// TwinCAT 3 PLC project Test_PLC_1
// ProgramVersion: 3.1.4024.0
// libraries:
//   Tc2_EtherCAT, * (Beckhoff Automation GmbH)
//   Tc2_Standard, * (Beckhoff Automation GmbH)
//   Tc2_System, * (Beckhoff Automation GmbH)
//   Tc3_Mc3PlanarMotion, * (Beckhoff Automation GmbH)
//   Tc3_Module, * (Beckhoff Automation GmbH)
//   Tc3_Physics, * (Beckhoff Automation GmbH)
//   Tc3_XPlanarStandard, * (Beckhoff Automation GmbH)
//   Tc3_XPlanarUtility, * (Beckhoff Automation GmbH)
//   VisuSymbols,3.5.10.0,System
// project tree:
//   DUTs/ ST_MoverParameters.TcDUT
//   / GlobalTextList.TcGTLO, PlcTask.TcTTO, Visualization Manager.TcVMO (not stored)
//   GVLs/ IO.TcGVL
//   POUs/Analytics/ CoeToPlc.TcPOU
//   POUs/ MAIN.TcPOU
//   POUs/xPlanar/ xPlanarControl.TcPOU, xPlanarProgram.TcPOU
//   VISUs/ Visualization.TcVIS
// real-time tasks:
//   TASK Job Task: cycle default, priority 32
//   TASK MC-Task (MET): cycle T#2ms, priority 10, ADS port 521
//   TASK MC-Task (MPT): cycle T#10ms, priority 18, ADS port 531
//   TASK PlcTask: cycle T#10ms, priority 20, ADS port 351
//   TASK XPlanar Task8: cycle T#250us, priority 4, ADS port 352
//   TASK XPlanar Task4: cycle T#250us, priority 6, ADS port 350
//   TASK PlcTask1: cycle T#10ms, priority 14, ADS port 353
// motion (NC):
//   TASK NC-Task 1 SAF: cycle T#2ms, priority 8, ADS port 501
//   TASK NC-Task 1 SVB: cycle T#10ms, priority 16, ADS port 511
//   AXIS Mover a-axis (id 2)
//     OtherSettings: AllowMotionCmdToSlave=true
//     encoder EncType=1
//     drive DrvType=5
//       Analog: TorqueSetpointScale=10, ScaleFactorActTorque=0.1
//       TimeComp: TaskDelayCycles=1
//     controller CtrType=1
//       CtrPara: PriorControlFactor=1
//         Observer: BandWidth=20
//   AXIS Mover b-axis (id 3)
//     OtherSettings: AllowMotionCmdToSlave=true
//     encoder EncType=1
//     drive DrvType=5
//       Analog: TorqueSetpointScale=10, ScaleFactorActTorque=0.1
//       TimeComp: TaskDelayCycles=1
//     controller CtrType=1
//       CtrPara: PriorControlFactor=1
//         Observer: BandWidth=20
//   AXIS Mover c-axis (id 4)
//     OtherSettings: AllowMotionCmdToSlave=true
//     encoder EncType=1
//     drive DrvType=5
//       Analog: TorqueSetpointScale=10, ScaleFactorActTorque=0.1
//       TimeComp: TaskDelayCycles=1
//     controller CtrType=1
//       CtrPara: PriorControlFactor=1
//         Observer: BandWidth=20
//   AXIS Mover x-axis (id 5)
//     OtherSettings: AllowMotionCmdToSlave=true
//     encoder EncType=1
//     drive DrvType=5
//       Analog: TorqueSetpointScale=10, ScaleFactorActTorque=0.1
//       TimeComp: TaskDelayCycles=1
//     controller CtrType=1
//       CtrPara: PriorControlFactor=1
//         Observer: BandWidth=20
//   AXIS Mover y-axis (id 6)
//     OtherSettings: AllowMotionCmdToSlave=true
//     encoder EncType=1
//     drive DrvType=5
//       Analog: TorqueSetpointScale=10, ScaleFactorActTorque=0.1
//       TimeComp: TaskDelayCycles=1
//     controller CtrType=1
//       CtrPara: PriorControlFactor=1
//         Observer: BandWidth=20
//   AXIS Mover z-axis (id 7)
//     OtherSettings: AllowMotionCmdToSlave=true
//     encoder EncType=1
//     drive DrvType=5
//       Analog: TorqueSetpointScale=10, ScaleFactorActTorque=0.1
//       TimeComp: TaskDelayCycles=1
//     controller CtrType=1
//       CtrPara: PriorControlFactor=1
//         Observer: BandWidth=20
// I/O:
//   DEVICE Device 1 (EtherCAT) (disabled), AmsNetId 192.168.5.90.2.1
//     Term 1 (EK1200) [EK1200-5000 EtherCAT Power supply (2A E-Bus)]
//       Term 2 (EL1004) [EL1004 4Ch. Dig. Input 24V, 3ms]
//       Term 3 (EL2004) [EL2004 4Ch. Dig. Output 24V, 0.5A]
//       Term 4 (EL9011) [EL9011 End Terminal]
//   DEVICE Device 4 (EtherCAT) (disabled), AmsNetId 192.168.5.90.7.1
//     Term 5 (APS4322-7000) [APS4322-7000 Drive]
//       Term 6 (APS4322-5000) [APS4322-5000 Feedback]
//     Term 7 (APS4322-7000) [APS4322-7000 Drive]
//       Term 8 (APS4322-5000) [APS4322-5000 Feedback]
// variable links:
//   Device 4 (EtherCAT) <-> TcCOM Objects/XPlanar/Part1/Tile1
//     Term 5 (APS4322-7000)/APS Comm Inputs/CommStatusWord <-> Data Pointer/MoverCommStatusWord
//     Term 5 (APS4322-7000)/APS Comm Inputs/Data {1..4} <-> Data Pointer/MoverCommDataIn[{0..3}]  (4 links)
//     Term 5 (APS4322-7000)/APS Comm Outputs/CommControlWord <-> Data Pointer/MoverCommControlWord
//     Term 5 (APS4322-7000)/APS Comm Outputs/Data 1 <-> Data Pointer/MoverCommDataOut
//     Term 5 (APS4322-7000)/APS Diagdata/DC Link Voltage <-> Data Pointer/DcLinkVoltage
//     Term 5 (APS4322-7000)/APS Diagdata/Power supply current <-> Data Pointer/PowerSupplyCurrent
//     Term 5 (APS4322-7000)/APS Inputs/StatusWord <-> Data Pointer/PowerUnitStatusWord
//     Term 5 (APS4322-7000)/APS Outputs/ControlWord <-> Data Pointer/PowerUnitControlWord
//     Term 5 (APS4322-7000)/APS Outputs/Current D 0X0 <-> Data Pointer/DCurrentSetPoints[0]
//     Term 5 (APS4322-7000)/APS Outputs/Current D 0X1 <-> Data Pointer/DCurrentSetPoints[1]
//     Term 5 (APS4322-7000)/APS Outputs/Current D 0X2 <-> Data Pointer/DCurrentSetPoints[2]
//     Term 5 (APS4322-7000)/APS Outputs/Current D 1X0 <-> Data Pointer/DCurrentSetPoints[6]
//     Term 5 (APS4322-7000)/APS Outputs/Current D 1X1 <-> Data Pointer/DCurrentSetPoints[7]
//     Term 5 (APS4322-7000)/APS Outputs/Current D 1X2 <-> Data Pointer/DCurrentSetPoints[8]
//     Term 5 (APS4322-7000)/APS Outputs/Current D 2X0 <-> Data Pointer/DCurrentSetPoints[12]
//     Term 5 (APS4322-7000)/APS Outputs/Current D 2X1 <-> Data Pointer/DCurrentSetPoints[13]
//     Term 5 (APS4322-7000)/APS Outputs/Current D 2X2 <-> Data Pointer/DCurrentSetPoints[14]
//     Term 5 (APS4322-7000)/APS Outputs/Current D 3X0 <-> Data Pointer/DCurrentSetPoints[18]
//     Term 5 (APS4322-7000)/APS Outputs/Current D 3X1 <-> Data Pointer/DCurrentSetPoints[19]
//     Term 5 (APS4322-7000)/APS Outputs/Current D 3X2 <-> Data Pointer/DCurrentSetPoints[20]
//     Term 5 (APS4322-7000)/APS Outputs/Current D 0Y0 <-> Data Pointer/DCurrentSetPoints[3]
//     Term 5 (APS4322-7000)/APS Outputs/Current D 0Y1 <-> Data Pointer/DCurrentSetPoints[4]
//     Term 5 (APS4322-7000)/APS Outputs/Current D 0Y2 <-> Data Pointer/DCurrentSetPoints[5]
//     Term 5 (APS4322-7000)/APS Outputs/Current D 1Y0 <-> Data Pointer/DCurrentSetPoints[9]
//     Term 5 (APS4322-7000)/APS Outputs/Current D 1Y1 <-> Data Pointer/DCurrentSetPoints[10]
//     Term 5 (APS4322-7000)/APS Outputs/Current D 1Y2 <-> Data Pointer/DCurrentSetPoints[11]
//     Term 5 (APS4322-7000)/APS Outputs/Current D 2Y0 <-> Data Pointer/DCurrentSetPoints[15]
//     Term 5 (APS4322-7000)/APS Outputs/Current D 2Y1 <-> Data Pointer/DCurrentSetPoints[16]
//     Term 5 (APS4322-7000)/APS Outputs/Current D 2Y2 <-> Data Pointer/DCurrentSetPoints[17]
//     Term 5 (APS4322-7000)/APS Outputs/Current D 3Y0 <-> Data Pointer/DCurrentSetPoints[21]
//     Term 5 (APS4322-7000)/APS Outputs/Current D 3Y1 <-> Data Pointer/DCurrentSetPoints[22]
//     Term 5 (APS4322-7000)/APS Outputs/Current D 3Y2 <-> Data Pointer/DCurrentSetPoints[23]
//     Term 5 (APS4322-7000)/APS Outputs/Current Q 0X0 <-> Data Pointer/QCurrentSetPoints[0]
//     Term 5 (APS4322-7000)/APS Outputs/Current Q 0X1 <-> Data Pointer/QCurrentSetPoints[1]
//     Term 5 (APS4322-7000)/APS Outputs/Current Q 0X2 <-> Data Pointer/QCurrentSetPoints[2]
//     Term 5 (APS4322-7000)/APS Outputs/Current Q 1X0 <-> Data Pointer/QCurrentSetPoints[6]
//     Term 5 (APS4322-7000)/APS Outputs/Current Q 1X1 <-> Data Pointer/QCurrentSetPoints[7]
//     Term 5 (APS4322-7000)/APS Outputs/Current Q 1X2 <-> Data Pointer/QCurrentSetPoints[8]
//     Term 5 (APS4322-7000)/APS Outputs/Current Q 2X0 <-> Data Pointer/QCurrentSetPoints[12]
//     Term 5 (APS4322-7000)/APS Outputs/Current Q 2X1 <-> Data Pointer/QCurrentSetPoints[13]
//     Term 5 (APS4322-7000)/APS Outputs/Current Q 2X2 <-> Data Pointer/QCurrentSetPoints[14]
//     Term 5 (APS4322-7000)/APS Outputs/Current Q 3X0 <-> Data Pointer/QCurrentSetPoints[18]
//     Term 5 (APS4322-7000)/APS Outputs/Current Q 3X1 <-> Data Pointer/QCurrentSetPoints[19]
//     Term 5 (APS4322-7000)/APS Outputs/Current Q 3X2 <-> Data Pointer/QCurrentSetPoints[20]
//     Term 5 (APS4322-7000)/APS Outputs/Current Q 0Y0 <-> Data Pointer/QCurrentSetPoints[3]
//     Term 5 (APS4322-7000)/APS Outputs/Current Q 0Y1 <-> Data Pointer/QCurrentSetPoints[4]
//     Term 5 (APS4322-7000)/APS Outputs/Current Q 0Y2 <-> Data Pointer/QCurrentSetPoints[5]
//     Term 5 (APS4322-7000)/APS Outputs/Current Q 1Y0 <-> Data Pointer/QCurrentSetPoints[9]
//     Term 5 (APS4322-7000)/APS Outputs/Current Q 1Y1 <-> Data Pointer/QCurrentSetPoints[10]
//     Term 5 (APS4322-7000)/APS Outputs/Current Q 1Y2 <-> Data Pointer/QCurrentSetPoints[11]
//     Term 5 (APS4322-7000)/APS Outputs/Current Q 2Y0 <-> Data Pointer/QCurrentSetPoints[15]
//     Term 5 (APS4322-7000)/APS Outputs/Current Q 2Y1 <-> Data Pointer/QCurrentSetPoints[16]
//     Term 5 (APS4322-7000)/APS Outputs/Current Q 2Y2 <-> Data Pointer/QCurrentSetPoints[17]
//     Term 5 (APS4322-7000)/APS Outputs/Current Q 3Y0 <-> Data Pointer/QCurrentSetPoints[21]
//     Term 5 (APS4322-7000)/APS Outputs/Current Q 3Y1 <-> Data Pointer/QCurrentSetPoints[22]
//     Term 5 (APS4322-7000)/APS Outputs/Current Q 3Y2 <-> Data Pointer/QCurrentSetPoints[23]
//     Term 5 (APS4322-7000)/APS Outputs/PhiE 0X0 <-> Data Pointer/PhiSetPoints[0]
//     Term 5 (APS4322-7000)/APS Outputs/PhiE 0X1 <-> Data Pointer/PhiSetPoints[1]
//     Term 5 (APS4322-7000)/APS Outputs/PhiE 0X2 <-> Data Pointer/PhiSetPoints[2]
//     Term 5 (APS4322-7000)/APS Outputs/PhiE 1X0 <-> Data Pointer/PhiSetPoints[6]
//     Term 5 (APS4322-7000)/APS Outputs/PhiE 1X1 <-> Data Pointer/PhiSetPoints[7]
//     Term 5 (APS4322-7000)/APS Outputs/PhiE 1X2 <-> Data Pointer/PhiSetPoints[8]
//     Term 5 (APS4322-7000)/APS Outputs/PhiE 2X0 <-> Data Pointer/PhiSetPoints[12]
//     Term 5 (APS4322-7000)/APS Outputs/PhiE 2X1 <-> Data Pointer/PhiSetPoints[13]
//     Term 5 (APS4322-7000)/APS Outputs/PhiE 2X2 <-> Data Pointer/PhiSetPoints[14]
//     Term 5 (APS4322-7000)/APS Outputs/PhiE 3X0 <-> Data Pointer/PhiSetPoints[18]
//     Term 5 (APS4322-7000)/APS Outputs/PhiE 3X1 <-> Data Pointer/PhiSetPoints[19]
//     Term 5 (APS4322-7000)/APS Outputs/PhiE 3X2 <-> Data Pointer/PhiSetPoints[20]
//     Term 5 (APS4322-7000)/APS Outputs/PhiE 0Y0 <-> Data Pointer/PhiSetPoints[3]
//     Term 5 (APS4322-7000)/APS Outputs/PhiE 0Y1 <-> Data Pointer/PhiSetPoints[4]
//     Term 5 (APS4322-7000)/APS Outputs/PhiE 0Y2 <-> Data Pointer/PhiSetPoints[5]
//     Term 5 (APS4322-7000)/APS Outputs/PhiE 1Y0 <-> Data Pointer/PhiSetPoints[9]
//     Term 5 (APS4322-7000)/APS Outputs/PhiE 1Y1 <-> Data Pointer/PhiSetPoints[10]
//     Term 5 (APS4322-7000)/APS Outputs/PhiE 1Y2 <-> Data Pointer/PhiSetPoints[11]
//     Term 5 (APS4322-7000)/APS Outputs/PhiE 2Y0 <-> Data Pointer/PhiSetPoints[15]
//     Term 5 (APS4322-7000)/APS Outputs/PhiE 2Y1 <-> Data Pointer/PhiSetPoints[16]
//     Term 5 (APS4322-7000)/APS Outputs/PhiE 2Y2 <-> Data Pointer/PhiSetPoints[17]
//     Term 5 (APS4322-7000)/APS Outputs/PhiE 3Y0 <-> Data Pointer/PhiSetPoints[21]
//     Term 5 (APS4322-7000)/APS Outputs/PhiE 3Y1 <-> Data Pointer/PhiSetPoints[22]
//     Term 5 (APS4322-7000)/APS Outputs/PhiE 3Y2 <-> Data Pointer/PhiSetPoints[23]
//     Term 5 (APS4322-7000)/Term 6 (APS4322-5000)/FB Inputs/A{0..8 step 2} X-Field <-> Data Pointer/HallSensorFieldsXYZ[{0..12 step 3}]  (5 links)
//     Term 5 (APS4322-7000)/Term 6 (APS4322-5000)/FB Inputs/A{0..8 step 2} Y-Field <-> Data Pointer/HallSensorFieldsXYZ[{1..13 step 3}]  (5 links)
//     Term 5 (APS4322-7000)/Term 6 (APS4322-5000)/FB Inputs/A{0..8 step 2} Z-Field <-> Data Pointer/HallSensorFieldsXYZ[{2..14 step 3}]  (5 links)
//     Term 5 (APS4322-7000)/Term 6 (APS4322-5000)/FB Inputs/B{1..9 step 2} X-Field <-> Data Pointer/HallSensorFieldsXYZ[{15..27 step 3}]  (5 links)
//     Term 5 (APS4322-7000)/Term 6 (APS4322-5000)/FB Inputs/B{1..9 step 2} Y-Field <-> Data Pointer/HallSensorFieldsXYZ[{16..28 step 3}]  (5 links)
//     Term 5 (APS4322-7000)/Term 6 (APS4322-5000)/FB Inputs/B{1..9 step 2} Z-Field <-> Data Pointer/HallSensorFieldsXYZ[{17..29 step 3}]  (5 links)
//     Term 5 (APS4322-7000)/Term 6 (APS4322-5000)/FB Inputs/C{0..8 step 2} X-Field <-> Data Pointer/HallSensorFieldsXYZ[{30..42 step 3}]  (5 links)
//     Term 5 (APS4322-7000)/Term 6 (APS4322-5000)/FB Inputs/C{0..8 step 2} Y-Field <-> Data Pointer/HallSensorFieldsXYZ[{31..43 step 3}]  (5 links)
//     Term 5 (APS4322-7000)/Term 6 (APS4322-5000)/FB Inputs/C{0..8 step 2} Z-Field <-> Data Pointer/HallSensorFieldsXYZ[{32..44 step 3}]  (5 links)
//     Term 5 (APS4322-7000)/Term 6 (APS4322-5000)/FB Inputs/D{1..9 step 2} X-Field <-> Data Pointer/HallSensorFieldsXYZ[{45..57 step 3}]  (5 links)
//     Term 5 (APS4322-7000)/Term 6 (APS4322-5000)/FB Inputs/D{1..9 step 2} Y-Field <-> Data Pointer/HallSensorFieldsXYZ[{46..58 step 3}]  (5 links)
//     Term 5 (APS4322-7000)/Term 6 (APS4322-5000)/FB Inputs/D{1..9 step 2} Z-Field <-> Data Pointer/HallSensorFieldsXYZ[{47..59 step 3}]  (5 links)
//     Term 5 (APS4322-7000)/Term 6 (APS4322-5000)/FB Inputs/E{0..8 step 2} X-Field <-> Data Pointer/HallSensorFieldsXYZ[{60..72 step 3}]  (5 links)
//     Term 5 (APS4322-7000)/Term 6 (APS4322-5000)/FB Inputs/E{0..8 step 2} Y-Field <-> Data Pointer/HallSensorFieldsXYZ[{61..73 step 3}]  (5 links)
//     Term 5 (APS4322-7000)/Term 6 (APS4322-5000)/FB Inputs/E{0..8 step 2} Z-Field <-> Data Pointer/HallSensorFieldsXYZ[{62..74 step 3}]  (5 links)
//     Term 5 (APS4322-7000)/Term 6 (APS4322-5000)/FB Inputs/F{1..9 step 2} X-Field <-> Data Pointer/HallSensorFieldsXYZ[{75..87 step 3}]  (5 links)
//     Term 5 (APS4322-7000)/Term 6 (APS4322-5000)/FB Inputs/F{1..9 step 2} Y-Field <-> Data Pointer/HallSensorFieldsXYZ[{76..88 step 3}]  (5 links)
//     Term 5 (APS4322-7000)/Term 6 (APS4322-5000)/FB Inputs/F{1..9 step 2} Z-Field <-> Data Pointer/HallSensorFieldsXYZ[{77..89 step 3}]  (5 links)
//     Term 5 (APS4322-7000)/Term 6 (APS4322-5000)/FB Inputs/G{0..8 step 2} X-Field <-> Data Pointer/HallSensorFieldsXYZ[{90..102 step 3}]  (5 links)
//     Term 5 (APS4322-7000)/Term 6 (APS4322-5000)/FB Inputs/G{0..8 step 2} Y-Field <-> Data Pointer/HallSensorFieldsXYZ[{91..103 step 3}]  (5 links)
//     Term 5 (APS4322-7000)/Term 6 (APS4322-5000)/FB Inputs/G{0..8 step 2} Z-Field <-> Data Pointer/HallSensorFieldsXYZ[{92..104 step 3}]  (5 links)
//     Term 5 (APS4322-7000)/Term 6 (APS4322-5000)/FB Inputs/H{1..9 step 2} X-Field <-> Data Pointer/HallSensorFieldsXYZ[{105..117 step 3}]  (5 links)
//     Term 5 (APS4322-7000)/Term 6 (APS4322-5000)/FB Inputs/H{1..9 step 2} Y-Field <-> Data Pointer/HallSensorFieldsXYZ[{106..118 step 3}]  (5 links)
//     Term 5 (APS4322-7000)/Term 6 (APS4322-5000)/FB Inputs/H{1..9 step 2} Z-Field <-> Data Pointer/HallSensorFieldsXYZ[{107..119 step 3}]  (5 links)
//     Term 5 (APS4322-7000)/Term 6 (APS4322-5000)/FB Inputs/I{0..8 step 2} X-Field <-> Data Pointer/HallSensorFieldsXYZ[{120..132 step 3}]  (5 links)
//     Term 5 (APS4322-7000)/Term 6 (APS4322-5000)/FB Inputs/I{0..8 step 2} Y-Field <-> Data Pointer/HallSensorFieldsXYZ[{121..133 step 3}]  (5 links)
//     Term 5 (APS4322-7000)/Term 6 (APS4322-5000)/FB Inputs/I{0..8 step 2} Z-Field <-> Data Pointer/HallSensorFieldsXYZ[{122..134 step 3}]  (5 links)
//     Term 5 (APS4322-7000)/Term 6 (APS4322-5000)/FB Inputs/J{1..9 step 2} X-Field <-> Data Pointer/HallSensorFieldsXYZ[{135..147 step 3}]  (5 links)
//     Term 5 (APS4322-7000)/Term 6 (APS4322-5000)/FB Inputs/J{1..9 step 2} Y-Field <-> Data Pointer/HallSensorFieldsXYZ[{136..148 step 3}]  (5 links)
//     Term 5 (APS4322-7000)/Term 6 (APS4322-5000)/FB Inputs/J{1..9 step 2} Z-Field <-> Data Pointer/HallSensorFieldsXYZ[{137..149 step 3}]  (5 links)
//     Term 5 (APS4322-7000)/Term 6 (APS4322-5000)/FB Inputs/Status <-> Data Pointer/FeedbackStatus
//   Device 4 (EtherCAT) <-> TcCOM Objects/XPlanar/Part1/Tile2
//     Term 7 (APS4322-7000)/APS Comm Inputs/CommStatusWord <-> Data Pointer/MoverCommStatusWord
//     Term 7 (APS4322-7000)/APS Comm Inputs/Data {1..4} <-> Data Pointer/MoverCommDataIn[{0..3}]  (4 links)
//     Term 7 (APS4322-7000)/APS Comm Outputs/CommControlWord <-> Data Pointer/MoverCommControlWord
//     Term 7 (APS4322-7000)/APS Comm Outputs/Data 1 <-> Data Pointer/MoverCommDataOut
//     Term 7 (APS4322-7000)/APS Diagdata/DC Link Voltage <-> Data Pointer/DcLinkVoltage
//     Term 7 (APS4322-7000)/APS Diagdata/Power supply current <-> Data Pointer/PowerSupplyCurrent
//     Term 7 (APS4322-7000)/APS Inputs/StatusWord <-> Data Pointer/PowerUnitStatusWord
//     Term 7 (APS4322-7000)/APS Outputs/ControlWord <-> Data Pointer/PowerUnitControlWord
//     Term 7 (APS4322-7000)/APS Outputs/Current D 0X0 <-> Data Pointer/DCurrentSetPoints[0]
//     Term 7 (APS4322-7000)/APS Outputs/Current D 0X1 <-> Data Pointer/DCurrentSetPoints[1]
//     Term 7 (APS4322-7000)/APS Outputs/Current D 0X2 <-> Data Pointer/DCurrentSetPoints[2]
//     Term 7 (APS4322-7000)/APS Outputs/Current D 1X0 <-> Data Pointer/DCurrentSetPoints[6]
//     Term 7 (APS4322-7000)/APS Outputs/Current D 1X1 <-> Data Pointer/DCurrentSetPoints[7]
//     Term 7 (APS4322-7000)/APS Outputs/Current D 1X2 <-> Data Pointer/DCurrentSetPoints[8]
//     Term 7 (APS4322-7000)/APS Outputs/Current D 2X0 <-> Data Pointer/DCurrentSetPoints[12]
//     Term 7 (APS4322-7000)/APS Outputs/Current D 2X1 <-> Data Pointer/DCurrentSetPoints[13]
//     Term 7 (APS4322-7000)/APS Outputs/Current D 2X2 <-> Data Pointer/DCurrentSetPoints[14]
//     Term 7 (APS4322-7000)/APS Outputs/Current D 3X0 <-> Data Pointer/DCurrentSetPoints[18]
//     Term 7 (APS4322-7000)/APS Outputs/Current D 3X1 <-> Data Pointer/DCurrentSetPoints[19]
//     Term 7 (APS4322-7000)/APS Outputs/Current D 3X2 <-> Data Pointer/DCurrentSetPoints[20]
//     Term 7 (APS4322-7000)/APS Outputs/Current D 0Y0 <-> Data Pointer/DCurrentSetPoints[3]
//     Term 7 (APS4322-7000)/APS Outputs/Current D 0Y1 <-> Data Pointer/DCurrentSetPoints[4]
//     Term 7 (APS4322-7000)/APS Outputs/Current D 0Y2 <-> Data Pointer/DCurrentSetPoints[5]
//     Term 7 (APS4322-7000)/APS Outputs/Current D 1Y0 <-> Data Pointer/DCurrentSetPoints[9]
//     Term 7 (APS4322-7000)/APS Outputs/Current D 1Y1 <-> Data Pointer/DCurrentSetPoints[10]
//     Term 7 (APS4322-7000)/APS Outputs/Current D 1Y2 <-> Data Pointer/DCurrentSetPoints[11]
//     Term 7 (APS4322-7000)/APS Outputs/Current D 2Y0 <-> Data Pointer/DCurrentSetPoints[15]
//     Term 7 (APS4322-7000)/APS Outputs/Current D 2Y1 <-> Data Pointer/DCurrentSetPoints[16]
//     Term 7 (APS4322-7000)/APS Outputs/Current D 2Y2 <-> Data Pointer/DCurrentSetPoints[17]
//     Term 7 (APS4322-7000)/APS Outputs/Current D 3Y0 <-> Data Pointer/DCurrentSetPoints[21]
//     Term 7 (APS4322-7000)/APS Outputs/Current D 3Y1 <-> Data Pointer/DCurrentSetPoints[22]
//     Term 7 (APS4322-7000)/APS Outputs/Current D 3Y2 <-> Data Pointer/DCurrentSetPoints[23]
//     Term 7 (APS4322-7000)/APS Outputs/Current Q 0X0 <-> Data Pointer/QCurrentSetPoints[0]
//     Term 7 (APS4322-7000)/APS Outputs/Current Q 0X1 <-> Data Pointer/QCurrentSetPoints[1]
//     Term 7 (APS4322-7000)/APS Outputs/Current Q 0X2 <-> Data Pointer/QCurrentSetPoints[2]
//     Term 7 (APS4322-7000)/APS Outputs/Current Q 1X0 <-> Data Pointer/QCurrentSetPoints[6]
//     Term 7 (APS4322-7000)/APS Outputs/Current Q 1X1 <-> Data Pointer/QCurrentSetPoints[7]
//     Term 7 (APS4322-7000)/APS Outputs/Current Q 1X2 <-> Data Pointer/QCurrentSetPoints[8]
//     Term 7 (APS4322-7000)/APS Outputs/Current Q 2X0 <-> Data Pointer/QCurrentSetPoints[12]
//     Term 7 (APS4322-7000)/APS Outputs/Current Q 2X1 <-> Data Pointer/QCurrentSetPoints[13]
//     Term 7 (APS4322-7000)/APS Outputs/Current Q 2X2 <-> Data Pointer/QCurrentSetPoints[14]
//     Term 7 (APS4322-7000)/APS Outputs/Current Q 3X0 <-> Data Pointer/QCurrentSetPoints[18]
//     Term 7 (APS4322-7000)/APS Outputs/Current Q 3X1 <-> Data Pointer/QCurrentSetPoints[19]
//     Term 7 (APS4322-7000)/APS Outputs/Current Q 3X2 <-> Data Pointer/QCurrentSetPoints[20]
//     Term 7 (APS4322-7000)/APS Outputs/Current Q 0Y0 <-> Data Pointer/QCurrentSetPoints[3]
//     Term 7 (APS4322-7000)/APS Outputs/Current Q 0Y1 <-> Data Pointer/QCurrentSetPoints[4]
//     Term 7 (APS4322-7000)/APS Outputs/Current Q 0Y2 <-> Data Pointer/QCurrentSetPoints[5]
//     Term 7 (APS4322-7000)/APS Outputs/Current Q 1Y0 <-> Data Pointer/QCurrentSetPoints[9]
//     Term 7 (APS4322-7000)/APS Outputs/Current Q 1Y1 <-> Data Pointer/QCurrentSetPoints[10]
//     Term 7 (APS4322-7000)/APS Outputs/Current Q 1Y2 <-> Data Pointer/QCurrentSetPoints[11]
//     Term 7 (APS4322-7000)/APS Outputs/Current Q 2Y0 <-> Data Pointer/QCurrentSetPoints[15]
//     Term 7 (APS4322-7000)/APS Outputs/Current Q 2Y1 <-> Data Pointer/QCurrentSetPoints[16]
//     Term 7 (APS4322-7000)/APS Outputs/Current Q 2Y2 <-> Data Pointer/QCurrentSetPoints[17]
//     Term 7 (APS4322-7000)/APS Outputs/Current Q 3Y0 <-> Data Pointer/QCurrentSetPoints[21]
//     Term 7 (APS4322-7000)/APS Outputs/Current Q 3Y1 <-> Data Pointer/QCurrentSetPoints[22]
//     Term 7 (APS4322-7000)/APS Outputs/Current Q 3Y2 <-> Data Pointer/QCurrentSetPoints[23]
//     Term 7 (APS4322-7000)/APS Outputs/PhiE 0X0 <-> Data Pointer/PhiSetPoints[0]
//     Term 7 (APS4322-7000)/APS Outputs/PhiE 0X1 <-> Data Pointer/PhiSetPoints[1]
//     Term 7 (APS4322-7000)/APS Outputs/PhiE 0X2 <-> Data Pointer/PhiSetPoints[2]
//     Term 7 (APS4322-7000)/APS Outputs/PhiE 1X0 <-> Data Pointer/PhiSetPoints[6]
//     Term 7 (APS4322-7000)/APS Outputs/PhiE 1X1 <-> Data Pointer/PhiSetPoints[7]
//     Term 7 (APS4322-7000)/APS Outputs/PhiE 1X2 <-> Data Pointer/PhiSetPoints[8]
//     Term 7 (APS4322-7000)/APS Outputs/PhiE 2X0 <-> Data Pointer/PhiSetPoints[12]
//     Term 7 (APS4322-7000)/APS Outputs/PhiE 2X1 <-> Data Pointer/PhiSetPoints[13]
//     Term 7 (APS4322-7000)/APS Outputs/PhiE 2X2 <-> Data Pointer/PhiSetPoints[14]
//     Term 7 (APS4322-7000)/APS Outputs/PhiE 3X0 <-> Data Pointer/PhiSetPoints[18]
//     Term 7 (APS4322-7000)/APS Outputs/PhiE 3X1 <-> Data Pointer/PhiSetPoints[19]
//     Term 7 (APS4322-7000)/APS Outputs/PhiE 3X2 <-> Data Pointer/PhiSetPoints[20]
//     Term 7 (APS4322-7000)/APS Outputs/PhiE 0Y0 <-> Data Pointer/PhiSetPoints[3]
//     Term 7 (APS4322-7000)/APS Outputs/PhiE 0Y1 <-> Data Pointer/PhiSetPoints[4]
//     Term 7 (APS4322-7000)/APS Outputs/PhiE 0Y2 <-> Data Pointer/PhiSetPoints[5]
//     Term 7 (APS4322-7000)/APS Outputs/PhiE 1Y0 <-> Data Pointer/PhiSetPoints[9]
//     Term 7 (APS4322-7000)/APS Outputs/PhiE 1Y1 <-> Data Pointer/PhiSetPoints[10]
//     Term 7 (APS4322-7000)/APS Outputs/PhiE 1Y2 <-> Data Pointer/PhiSetPoints[11]
//     Term 7 (APS4322-7000)/APS Outputs/PhiE 2Y0 <-> Data Pointer/PhiSetPoints[15]
//     Term 7 (APS4322-7000)/APS Outputs/PhiE 2Y1 <-> Data Pointer/PhiSetPoints[16]
//     Term 7 (APS4322-7000)/APS Outputs/PhiE 2Y2 <-> Data Pointer/PhiSetPoints[17]
//     Term 7 (APS4322-7000)/APS Outputs/PhiE 3Y0 <-> Data Pointer/PhiSetPoints[21]
//     Term 7 (APS4322-7000)/APS Outputs/PhiE 3Y1 <-> Data Pointer/PhiSetPoints[22]
//     Term 7 (APS4322-7000)/APS Outputs/PhiE 3Y2 <-> Data Pointer/PhiSetPoints[23]
//     Term 7 (APS4322-7000)/Term 8 (APS4322-5000)/FB Inputs/A{0..8 step 2} X-Field <-> Data Pointer/HallSensorFieldsXYZ[{0..12 step 3}]  (5 links)
//     Term 7 (APS4322-7000)/Term 8 (APS4322-5000)/FB Inputs/A{0..8 step 2} Y-Field <-> Data Pointer/HallSensorFieldsXYZ[{1..13 step 3}]  (5 links)
//     Term 7 (APS4322-7000)/Term 8 (APS4322-5000)/FB Inputs/A{0..8 step 2} Z-Field <-> Data Pointer/HallSensorFieldsXYZ[{2..14 step 3}]  (5 links)
//     Term 7 (APS4322-7000)/Term 8 (APS4322-5000)/FB Inputs/B{1..9 step 2} X-Field <-> Data Pointer/HallSensorFieldsXYZ[{15..27 step 3}]  (5 links)
//     Term 7 (APS4322-7000)/Term 8 (APS4322-5000)/FB Inputs/B{1..9 step 2} Y-Field <-> Data Pointer/HallSensorFieldsXYZ[{16..28 step 3}]  (5 links)
//     Term 7 (APS4322-7000)/Term 8 (APS4322-5000)/FB Inputs/B{1..9 step 2} Z-Field <-> Data Pointer/HallSensorFieldsXYZ[{17..29 step 3}]  (5 links)
//     Term 7 (APS4322-7000)/Term 8 (APS4322-5000)/FB Inputs/C{0..8 step 2} X-Field <-> Data Pointer/HallSensorFieldsXYZ[{30..42 step 3}]  (5 links)
//     Term 7 (APS4322-7000)/Term 8 (APS4322-5000)/FB Inputs/C{0..8 step 2} Y-Field <-> Data Pointer/HallSensorFieldsXYZ[{31..43 step 3}]  (5 links)
//     Term 7 (APS4322-7000)/Term 8 (APS4322-5000)/FB Inputs/C{0..8 step 2} Z-Field <-> Data Pointer/HallSensorFieldsXYZ[{32..44 step 3}]  (5 links)
//     Term 7 (APS4322-7000)/Term 8 (APS4322-5000)/FB Inputs/D{1..9 step 2} X-Field <-> Data Pointer/HallSensorFieldsXYZ[{45..57 step 3}]  (5 links)
//     Term 7 (APS4322-7000)/Term 8 (APS4322-5000)/FB Inputs/D{1..9 step 2} Y-Field <-> Data Pointer/HallSensorFieldsXYZ[{46..58 step 3}]  (5 links)
//     Term 7 (APS4322-7000)/Term 8 (APS4322-5000)/FB Inputs/D{1..9 step 2} Z-Field <-> Data Pointer/HallSensorFieldsXYZ[{47..59 step 3}]  (5 links)
//     Term 7 (APS4322-7000)/Term 8 (APS4322-5000)/FB Inputs/E{0..8 step 2} X-Field <-> Data Pointer/HallSensorFieldsXYZ[{60..72 step 3}]  (5 links)
//     Term 7 (APS4322-7000)/Term 8 (APS4322-5000)/FB Inputs/E{0..8 step 2} Y-Field <-> Data Pointer/HallSensorFieldsXYZ[{61..73 step 3}]  (5 links)
//     Term 7 (APS4322-7000)/Term 8 (APS4322-5000)/FB Inputs/E{0..8 step 2} Z-Field <-> Data Pointer/HallSensorFieldsXYZ[{62..74 step 3}]  (5 links)
//     Term 7 (APS4322-7000)/Term 8 (APS4322-5000)/FB Inputs/F{1..9 step 2} X-Field <-> Data Pointer/HallSensorFieldsXYZ[{75..87 step 3}]  (5 links)
//     Term 7 (APS4322-7000)/Term 8 (APS4322-5000)/FB Inputs/F{1..9 step 2} Y-Field <-> Data Pointer/HallSensorFieldsXYZ[{76..88 step 3}]  (5 links)
//     Term 7 (APS4322-7000)/Term 8 (APS4322-5000)/FB Inputs/F{1..9 step 2} Z-Field <-> Data Pointer/HallSensorFieldsXYZ[{77..89 step 3}]  (5 links)
//     Term 7 (APS4322-7000)/Term 8 (APS4322-5000)/FB Inputs/G{0..8 step 2} X-Field <-> Data Pointer/HallSensorFieldsXYZ[{90..102 step 3}]  (5 links)
//     Term 7 (APS4322-7000)/Term 8 (APS4322-5000)/FB Inputs/G{0..8 step 2} Y-Field <-> Data Pointer/HallSensorFieldsXYZ[{91..103 step 3}]  (5 links)
//     Term 7 (APS4322-7000)/Term 8 (APS4322-5000)/FB Inputs/G{0..8 step 2} Z-Field <-> Data Pointer/HallSensorFieldsXYZ[{92..104 step 3}]  (5 links)
//     Term 7 (APS4322-7000)/Term 8 (APS4322-5000)/FB Inputs/H{1..9 step 2} X-Field <-> Data Pointer/HallSensorFieldsXYZ[{105..117 step 3}]  (5 links)
//     Term 7 (APS4322-7000)/Term 8 (APS4322-5000)/FB Inputs/H{1..9 step 2} Y-Field <-> Data Pointer/HallSensorFieldsXYZ[{106..118 step 3}]  (5 links)
//     Term 7 (APS4322-7000)/Term 8 (APS4322-5000)/FB Inputs/H{1..9 step 2} Z-Field <-> Data Pointer/HallSensorFieldsXYZ[{107..119 step 3}]  (5 links)
//     Term 7 (APS4322-7000)/Term 8 (APS4322-5000)/FB Inputs/I{0..8 step 2} X-Field <-> Data Pointer/HallSensorFieldsXYZ[{120..132 step 3}]  (5 links)
//     Term 7 (APS4322-7000)/Term 8 (APS4322-5000)/FB Inputs/I{0..8 step 2} Y-Field <-> Data Pointer/HallSensorFieldsXYZ[{121..133 step 3}]  (5 links)
//     Term 7 (APS4322-7000)/Term 8 (APS4322-5000)/FB Inputs/I{0..8 step 2} Z-Field <-> Data Pointer/HallSensorFieldsXYZ[{122..134 step 3}]  (5 links)
//     Term 7 (APS4322-7000)/Term 8 (APS4322-5000)/FB Inputs/J{1..9 step 2} X-Field <-> Data Pointer/HallSensorFieldsXYZ[{135..147 step 3}]  (5 links)
//     Term 7 (APS4322-7000)/Term 8 (APS4322-5000)/FB Inputs/J{1..9 step 2} Y-Field <-> Data Pointer/HallSensorFieldsXYZ[{136..148 step 3}]  (5 links)
//     Term 7 (APS4322-7000)/Term 8 (APS4322-5000)/FB Inputs/J{1..9 step 2} Z-Field <-> Data Pointer/HallSensorFieldsXYZ[{137..149 step 3}]  (5 links)
//     Term 7 (APS4322-7000)/Term 8 (APS4322-5000)/FB Inputs/Status <-> Data Pointer/FeedbackStatus
//   XPlanar MC Project/Axes/Mover4220_1 <-> TcCOM Objects/XPlanar/Mover4220_1
//     McToIo/STD <-> InputsFromNC3/NC3ToHW
//   XPlanar MC Project/Axes/Mover4220_2 <-> TcCOM Objects/XPlanar/Mover4220_2
//     McToIo/STD <-> InputsFromNC3/NC3ToHW
//   Test PLC 1/Test PLC 1 Instance <-> Device 1 (EtherCAT)/Term 1 (EK1200)/Term 2 (EL1004)
//     PlcTask Inputs/IO.HardwareInput[{1..4}] <-> Channel {1..4}/Input  (4 links)
//   Test PLC 1/Test PLC 1 Instance <-> Device 1 (EtherCAT)/Term 1 (EK1200)/Term 3 (EL2004)
//     PlcTask Outputs/IO.HardwareOutput[{1..4}] <-> Channel {1..4}/Output  (4 links)
//   Test PLC 1/Test PLC 1 Instance <-> XPlanar MC Project/Axes/Mover4220_1
//     PlcTask Inputs/xPlanarProgram.xPlanar._PlanarMover[1].MCTOPLC/ACT <-> McToPlc/ACT
//     PlcTask Inputs/xPlanarProgram.xPlanar._PlanarMover[1].MCTOPLC/COORDMODE <-> McToPlc/COORDMODE
//     PlcTask Inputs/xPlanarProgram.xPlanar._PlanarMover[1].MCTOPLC/SET <-> McToPlc/SET
//     PlcTask Inputs/xPlanarProgram.xPlanar._PlanarMover[1].MCTOPLC/SETONTRACK <-> McToPlc/SETONTRACK
//     PlcTask Inputs/xPlanarProgram.xPlanar._PlanarMover[1].MCTOPLC/STD <-> McToPlc/STD
//     PlcTask Outputs/xPlanarProgram.xPlanar._PlanarMover[1].PLCTOMC/STD <-> PlcToMc/STD
//   Test PLC 1/Test PLC 1 Instance <-> XPlanar MC Project/Axes/Mover4220_2
//     PlcTask Inputs/xPlanarProgram.xPlanar._PlanarMover[2].MCTOPLC/ACT <-> McToPlc/ACT
//     PlcTask Inputs/xPlanarProgram.xPlanar._PlanarMover[2].MCTOPLC/COORDMODE <-> McToPlc/COORDMODE
//     PlcTask Inputs/xPlanarProgram.xPlanar._PlanarMover[2].MCTOPLC/SET <-> McToPlc/SET
//     PlcTask Inputs/xPlanarProgram.xPlanar._PlanarMover[2].MCTOPLC/SETONTRACK <-> McToPlc/SETONTRACK
//     PlcTask Inputs/xPlanarProgram.xPlanar._PlanarMover[2].MCTOPLC/STD <-> McToPlc/STD
//     PlcTask Outputs/xPlanarProgram.xPlanar._PlanarMover[2].PLCTOMC/STD <-> PlcToMc/STD
//   Test PLC 1/Test PLC 1 Instance <-> XPlanar MC Project/Groups/Environment
//     PlcTask Inputs/xPlanarProgram.xPlanar._PlanarEnvironment.MCTOPLC_STD <-> McToPlc/STD
//   Test PLC 1/Test PLC 1 Instance <-> XPlanar MC Project/Groups/XPlanar
//     PlcTask Inputs/xPlanarProgram.xPlanar._PlanarGroup.MCTOPLC_STD <-> McToPlc/STD
//   TcCOM Objects/XPlanar/Mover4220_1 <-> XPlanar MC Project/Axes/Mover4220_1
//     OutputsToNC3/HWToNC3 <-> IoToMc/STD
//   TcCOM Objects/XPlanar/Mover4220_2 <-> XPlanar MC Project/Axes/Mover4220_2
//     OutputsToNC3/HWToNC3 <-> IoToMc/STD

CONFIGURATION Test_PLC_1
    RESOURCE PLC ON TwinCAT3
        TASK PlcTask(INTERVAL := T#10ms, PRIORITY := 14);
        PROGRAM MAIN WITH PlcTask : MAIN;
    END_RESOURCE
END_CONFIGURATION

// ---- DUTs/ST_MoverParameters.TcDUT
TYPE ST_MoverParameters :
STRUCT
	sLogMessage			:	STRING;
	targetPosition		:	PositionXYC;
	Constraints			:	DynamicConstraint_PathXY;
	Options				:	ST_MoveToPositionOptions;
	rotateOptions		:	ST_MoveCOptions;
	rotateSetPosition	: 	LREAL;
	joinTrackOptions	:	ST_JoinTrackOptions;
	leaveTrackOptions	:	ST_LeaveTrackOptions;
	extPosModeOptions	:	MC_EXTERNAL_SET_POSITION_MODE;
END_STRUCT
END_TYPE

// ---- GVLs/IO.TcGVL
{attribute 'qualified_only'}
VAR_GLOBAL
	HardwareInput		AT %I* : ARRAY [1..4] OF BOOL;
	HardwareOutput		AT %Q* : ARRAY [1..4] OF BOOL;
END_VAR

// ---- POUs/MAIN.TcPOU
PROGRAM MAIN
VAR
	Running				: BYTE;
	TimeAlive			: TON;
	TimeAliveSeconds	: INT;

END_VAR



// ======================================================================== //
//																			//
//					Beckhoff 2-Tile xPlanar Program							//
//																			//
//					Last Updated: 19-MAR-2025								//
//					Last Programmer: Ben Sturdy								//
//																			//
// ======================================================================== //


Running := Running + 1;


// Time the system has been in run mode (in seconds)
TimeAlive(IN := NOT TimeAlive.Q, PT := T#1S);
IF TimeAlive.Q THEN
	TimeAliveSeconds := TimeAliveSeconds + 1;
END_IF


xPlanarProgram();


CoeToPlc();

END_PROGRAM

// ---- POUs/xPlanar/xPlanarProgram.TcPOU
PROGRAM xPlanarProgram
VAR
	
	xPlanar			: xPlanarControl;
	
	State			: BYTE;
	
	ProgramTrigger	: R_Trig;
	LEDTimer		: TON;

	FlashTime		: TIME := T#250MS;
	
	ProgramRunning	: BOOL;
	
END_VAR




















// ---------- LED logic

ProgramTrigger(CLK := IO.HardwareInput[1]);
LEDTimer(IN := (NOT(LEDTimer.Q)), PT := FlashTime);

IF LEDTimer.Q THEN
	IO.HardwareOutput[1] := NOT(IO.HardwareOutput[1]);
END_IF

IF ProgramTrigger.Q THEN
	ProgramRunning := NOT(ProgramRunning);
END_IF

IF (NOT(ProgramRunning) AND (State <> 0)) THEN
	FlashTime := T#200MS;
ELSE
	FlashTime := T#1000MS;
END_IF



// ---------- xPlanar control program

xPlanar.CyclicUpdate();

IF xPlanar.DetectErrors() THEN
	State := 99;
END_IF

CASE State OF
	
	0:
		IF ProgramRunning THEN
			State := 1;
		ELSE
			State := 0;
		END_IF
		
	1:	
		IF xPlanar.EnableMovers() THEN
			State := 2;
		END_IF
		
	{66:}
		IF xPlanar.CaEnable() THEN
			State := 2;
		END_IF}
		
	2:
		IF ProgramRunning THEN
			State := 3;
		ELSE
			State := 0;
		END_IF
		
	3:
		IF xPlanar.Home() THEN
			State := 4;
		END_IF
		
	4:
		IF ProgramRunning THEN
			State := 5;
		ELSE
			State := 0;
		END_IF
		
	5:
		IF xPlanar.SwapPlaces() THEN
			State := 6;
		END_IF	
		
	6:
		IF ProgramRunning THEN
			State := 7;
		ELSE
			State := 0;
		END_IF
		
	7:
		IF xPlanar.FollowTileEdge() THEN
			State := 8;
		END_IF
		
	8:
		IF ProgramRunning THEN
			State := 9;
		ELSE
			State := 0;
		END_IF
		
	9:
		IF xPlanar.VaryMoverHeight() THEN
			State := 10;
		END_IF
		
	10:
		IF ProgramRunning THEN
			State := 11;
		ELSE
			State := 0;
		END_IF
		
	11:
		IF xPlanar.Spin() THEN
			State := 12;
		END_IF
		
	12:
		IF ProgramRunning THEN
			State := 13;
		ELSE
			State := 0;
		END_IF
		
	13:
		IF xPlanar.Tilt() THEN
			State := 2;
		END_IF
			
	99:
		IF xPlanar.ResetErrors() THEN
			State := 0;
		END_IF	
	
END_CASE

END_PROGRAM

// ---- POUs/xPlanar/xPlanarControl.TcPOU
FUNCTION_BLOCK xPlanarControl
VAR
	
	// xPlanar objects
	_PlanarMover				: ARRAY [1.._MoverCount] OF MC_PlanarMover;
	_PlanarMoverFeedback		: ARRAY [1.._MoverCount] OF MC_PlanarFeedback;
	_PlanarGroup				: MC_PlanarGroup;
	_PlanarGroupFeedback		: MC_PlanarFeedback;
	_PlanarEnvironment			: MC_PlanarEnvironment;
	_PlanarEnvironmentFeedback	: MC_PlanarFeedback;
	_PlanarTrack				: ARRAY [1.._TrackCount] OF MC_PlanarTrack;
	_PlanarTrackFeedback		: ARRAY [1.._TrackCount] OF MC_PlanarFeedback;
	
	_MoveParameters				: ARRAY [1.._MoverCount] OF ST_MoverParameters;
	
	// Internal states and counters
	_i							: UINT := 0;
	_LocalState					: UINT := 0;
	_InternalCounter			: UINT := 0;
	_ErrorCount					: UINT := 0;
	_CommandDone				: BOOL := FALSE;
	
	// Status of movers
	_Enabled					: ARRAY [1.._MoverCount] OF BOOL;
	_Error						: ARRAY [1.._MoverCount] OF BOOL;
	_ErrorCode					: ARRAY [1.._MoverCount] OF UDINT;
	_ErrorCodePrevious			: ARRAY [1.._MoverCount] OF UDINT;
	_Busy						: ARRAY [1.._MoverCount] OF BOOL;
	_Done						: ARRAY [1.._MoverCount] OF BOOL;
	
	// Parameters of movers
	_Velocity					: LREAL := 2000;
	_Acceleration				: LREAL := 20000;
	_Deceleration				: LREAL := 20000;
	_Jerk						: LREAL := 200000;
	_NumberOfRotations			: UDINT := 5;
	
END_VAR
VAR CONSTANT
	
	// Number of movers
	_MoverCount					: UINT := 2;
	_TrackCount					: UINT := 3;

END_VAR

// NETWORK 1

METHOD CaAddAllMoversToGroup : BOOL
VAR_INPUT
END_VAR
// Enable planar group and add all movers

CASE _LocalState OF
	
	0:
		_LocalState := 1;

	1:
		FOR _i := 1 TO _MoverCount DO
			_PlanarMover[_i].AddToGroup
			(
				commandFeedback := _PlanarMoverFeedback[_i],
				group := _PlanarGroup
			);
		END_FOR
		_LocalState := 2;
	
	2:
		_CommandDone := TRUE;
		FOR _i := 1 TO _MoverCount DO
			IF NOT(_PlanarMoverFeedback[_i].Done) THEN
				_CommandDone := FALSE;
				_InternalCounter := _InternalCounter + 1;
			END_IF
		END_FOR
		
		IF _InternalCounter >= 10000 THEN
			_LocalState := 0;
			_InternalCounter := 0;
			CaAddAllMoversToGroup := FALSE;
		END_IF
		
		IF _CommandDone THEN
			_CommandDone := FALSE;
			_InternalCounter := 0;
			_LocalState := 3;
		END_IF
	
	3:
		_LocalState := 0;
		CaAddAllMoversToGroup := TRUE;
		
END_CASE
END_METHOD

METHOD CaDisable : BOOL
VAR_INPUT
END_VAR

// Enable planar group and add all movers

CASE _LocalState OF
	
	0:
		_LocalState := 1;

	1:
		_PlanarGroup.Disable(commandFeedback := _PlanarGroupFeedback);
		_LocalState := 2;
	
	2:
		IF _PlanarGroupFeedback.Done THEN
			_LocalState := 3;
		END_IF
	
	3:
		_LocalState := 0;
		CaDisable := TRUE;
		
END_CASE
END_METHOD

METHOD CaEnable : BOOL
VAR_INPUT
END_VAR

// Enable planar group and add all movers

CASE _LocalState OF
	
	0:
		_LocalState := 1;

	1:
		_PlanarGroup.Enable(commandFeedback := _PlanarGroupFeedback);
		_LocalState := 2;
	
	2:
		IF _PlanarGroupFeedback.Done THEN
			_LocalState := 3;
		END_IF
	
	3:
		_LocalState := 0;
		CaEnable := TRUE;
		
END_CASE
END_METHOD

METHOD CyclicUpdate : BOOL
VAR_INPUT
END_VAR


// Update method needs to be called cyclically


_PlanarGroup.Update();
_PlanarGroupFeedback.Update();


FOR _i := 1 TO _MoverCount DO
	

	_PlanarMover[_i].Update();
	_PlanarMoverFeedback[_i].Update();
		
	
	IF _PlanarMover[_i].MCTOPLC.STD.State = 3 THEN
		_Enabled[_i] := TRUE;
	ELSE
		_Enabled[_i] := FALSE;
	END_IF
	

	_Error[_i] := _PlanarMoverFeedback[_i].Error;
	_Busy[_i] := _PlanarMoverFeedback[_i].Busy;
	_Done[_i] := _PlanarMoverFeedback[_i].Done;
	_ErrorCode[_i] := _PlanarMoverFeedback[_i].ErrorId;
	IF _PlanarMoverFeedback[_i].ErrorId <> 0 THEN
		_ErrorCodePrevious[_i] := _PlanarMoverFeedback[_i].ErrorId;
	END_IF
	
	
	_MoveParameters[_i].Options.useOrientation := TRUE;
	_MoveParameters[_i].Constraints.SetValuesVADJ(V := _Velocity, A := _Acceleration, D := _Deceleration, J := _Jerk);
	_MoveParameters[_i].rotateOptions.additionalTurns := _NumberOfRotations;
	
	
	_MoveParameters[_i].Constraints
	
	
	IF (_i MOD 2 <> 0) THEN
		_MoveParameters[_i].rotateOptions.direction := 1;
	ELSE
		_MoveParameters[_i].rotateOptions.direction := 3;
	END_IF
	
	
END_FOR
END_METHOD

METHOD PUBLIC DecreaseMoverHeight : BOOL
VAR_INPUT
END_VAR

// Movers decrease height
	
CASE _LocalState OF
	
	0:
		_LocalState := 1;
	
	1:
		FOR _i := 1 TO _MoverCount DO
			_PlanarMover[_i].MoveZ
			(	
				commandFeedback		:= _PlanarMoverFeedback[_i],
				targetPosition		:= 2.0,
				constraint			:= _MoveParameters[_i].Constraints
			);
		END_FOR
		_LocalState := 2;
	
	2:
		_CommandDone := TRUE;
		FOR _i := 1 TO _MoverCount DO
			IF NOT(_PlanarMoverFeedback[_i].Done) THEN
				_CommandDone := FALSE;
				_InternalCounter := _InternalCounter + 1;
			END_IF
		END_FOR
		
		IF _InternalCounter >= 10000 THEN
			_LocalState := 0;
			_InternalCounter := 0;
			DecreaseMoverHeight := FALSE;
		END_IF
		
		IF _CommandDone THEN
			_CommandDone := FALSE;
			_InternalCounter := 0;
			_LocalState := 2;
		END_IF

	3:
		DecreaseMoverHeight := TRUE;
		_LocalState := 0;

END_CASE
END_METHOD

METHOD DetectErrors : BOOL
VAR_INPUT
END_VAR


// Error detection method

FOR _i := 1 TO _MoverCount DO
	IF _PlanarMover[_i].Error THEN
		_Error[_i] := TRUE;
		_LocalState := 0;
		_InternalCounter := 0;
		DetectErrors := TRUE;
	END_IF
END_FOR
END_METHOD

METHOD DisableMovers : BOOL
VAR_INPUT
END_VAR


// Disable movers

CASE _LocalState OF
	
	0:
		FOR _i := 1 TO _MoverCount DO
			_PlanarMover[_i].Disable(_PlanarMoverFeedback[_i]);
		END_FOR
		_LocalState := 1;
	
	1:
		_CommandDone := TRUE;
		FOR _i := 1 TO _MoverCount DO
			IF NOT(_PlanarMoverFeedback[_i].Done) THEN
				_CommandDone := FALSE;
				_InternalCounter := _InternalCounter + 1;
			END_IF
		END_FOR
		
		IF _InternalCounter >= 10000 THEN
			_LocalState := 0;
			_InternalCounter := 0;
			DisableMovers := FALSE;
		END_IF
		
		IF _CommandDone THEN
			_CommandDone := FALSE;
			_InternalCounter := 0;
			_LocalState := 2;
		END_IF
	
	2:
		_LocalState := 0;
		DisableMovers := TRUE;

END_CASE
END_METHOD

METHOD EnableMovers : BOOL
VAR_INPUT
END_VAR


// Enable movers

CASE _LocalState OF
	
	0:
		FOR _i := 1 TO _MoverCount DO
			_PlanarMover[_i].Enable(_PlanarMoverFeedback[_i]);
		END_FOR
		_LocalState := 1;
	
	1:
		_CommandDone := TRUE;
		FOR _i := 1 TO _MoverCount DO
			IF NOT(_PlanarMoverFeedback[_i].Done) THEN
				_CommandDone := FALSE;
				_InternalCounter := _InternalCounter + 1;
			END_IF
		END_FOR
		
		IF _InternalCounter >= 10000 THEN
			_LocalState := 0;
			_InternalCounter := 0;
			EnableMovers := FALSE;
		END_IF
		
		IF _CommandDone THEN
			_CommandDone := FALSE;
			_InternalCounter := 0;
			_LocalState := 2;
		END_IF
	
	2:
		_LocalState := 0;
		EnableMovers := TRUE;

END_CASE
END_METHOD

METHOD PUBLIC FollowTileEdge : BOOL
VAR_INPUT
END_VAR
// Movers move to edge of tiles and follow the perimeter, then move to home
	
CASE _LocalState OF
	
	0:
		_LocalState := 1;

	1:
		_MoveParameters[1].targetPosition.x := 180;
		_MoveParameters[1].targetPosition.y := 183;
		_MoveParameters[2].targetPosition.x := 296;
		_MoveParameters[2].targetPosition.y := 183;
		_LocalState := 2;
	
	2:
		FOR _i := 1 TO _MoverCount DO
			_PlanarMover[_i].MoveToPosition
			(
				commandFeedback 	:= _PlanarMoverFeedback[_i],
				targetPosition 		:= _MoveParameters[_i].targetPosition,
				constraint 			:= _MoveParameters[_i].Constraints,
				options 			:= _MoveParameters[_i].Options
			);
		END_FOR
		_LocalState := 3;
	
	3:
		_CommandDone := TRUE;
		FOR _i := 1 TO _MoverCount DO
			IF NOT(_PlanarMoverFeedback[_i].Done) THEN
				_CommandDone := FALSE;
				_InternalCounter := _InternalCounter + 1;
			END_IF
		END_FOR
		
		IF _InternalCounter >= 10000 THEN
			_LocalState := 0;
			_InternalCounter := 0;
			FollowTileEdge := FALSE;
		END_IF
		
		IF _CommandDone THEN
			_CommandDone := FALSE;
			_InternalCounter := 0;
			_LocalState := 4;
		END_IF

	4:
		_MoveParameters[1].targetPosition.x := 57;
		_MoveParameters[1].targetPosition.y := 183;
		_MoveParameters[2].targetPosition.x := 423;
		_MoveParameters[2].targetPosition.y := 183;
		_LocalState := 5;
	
	5:
		FOR _i := 1 TO _MoverCount DO
			_PlanarMover[_i].MoveToPosition
			(
				commandFeedback 	:= _PlanarMoverFeedback[_i],
				targetPosition 		:= _MoveParameters[_i].targetPosition,
				constraint 			:= _MoveParameters[_i].Constraints,
				options 			:= _MoveParameters[_i].Options
			);
		END_FOR
		_LocalState := 6;
	
	6:
		_CommandDone := TRUE;
		FOR _i := 1 TO _MoverCount DO
			IF NOT(_PlanarMoverFeedback[_i].Done) THEN
				_CommandDone := FALSE;
				_InternalCounter := _InternalCounter + 1;
			END_IF
		END_FOR
		
		IF _InternalCounter >= 10000 THEN
			_LocalState := 0;
			_InternalCounter := 0;
			FollowTileEdge := FALSE;
		END_IF
		
		IF _CommandDone THEN
			_CommandDone := FALSE;
			_InternalCounter := 0;
			_LocalState := 7;
		END_IF
		
	7:
		_MoveParameters[1].targetPosition.x := 57;
		_MoveParameters[1].targetPosition.y := 57;
		_MoveParameters[2].targetPosition.x := 423;
		_MoveParameters[2].targetPosition.y := 57;
		_LocalState := 8;
	
	8:
		FOR _i := 1 TO _MoverCount DO
			_PlanarMover[_i].MoveToPosition
			(
				commandFeedback 	:= _PlanarMoverFeedback[_i],
				targetPosition 		:= _MoveParameters[_i].targetPosition,
				constraint 			:= _MoveParameters[_i].Constraints,
				options 			:= _MoveParameters[_i].Options
			);
		END_FOR
		_LocalState := 9;
	
	9:
		_CommandDone := TRUE;
		FOR _i := 1 TO _MoverCount DO
			IF NOT(_PlanarMoverFeedback[_i].Done) THEN
				_CommandDone := FALSE;
				_InternalCounter := _InternalCounter + 1;
			END_IF
		END_FOR
		
		IF _InternalCounter >= 10000 THEN
			_LocalState := 0;
			_InternalCounter := 0;
			FollowTileEdge := FALSE;
		END_IF
		
		IF _CommandDone THEN
			_CommandDone := FALSE;
			_InternalCounter := 0;
			_LocalState := 10;
		END_IF
		
	10:
		_MoveParameters[1].targetPosition.x := 180;
		_MoveParameters[1].targetPosition.y := 57;
		_MoveParameters[2].targetPosition.x := 296;
		_MoveParameters[2].targetPosition.y := 57;
		_LocalState := 11;
	
	11:
		FOR _i := 1 TO _MoverCount DO
			_PlanarMover[_i].MoveToPosition
			(
				commandFeedback 	:= _PlanarMoverFeedback[_i],
				targetPosition 		:= _MoveParameters[_i].targetPosition,
				constraint 			:= _MoveParameters[_i].Constraints,
				options 			:= _MoveParameters[_i].Options
			);
		END_FOR
		_LocalState := 12;
	
	12:
		_CommandDone := TRUE;
		FOR _i := 1 TO _MoverCount DO
			IF NOT(_PlanarMoverFeedback[_i].Done) THEN
				_CommandDone := FALSE;
				_InternalCounter := _InternalCounter + 1;
			END_IF
		END_FOR
		
		IF _InternalCounter >= 10000 THEN
			_LocalState := 0;
			_InternalCounter := 0;
			FollowTileEdge := FALSE;
		END_IF
		
		IF _CommandDone THEN
			_CommandDone := FALSE;
			_InternalCounter := 0;
			_LocalState := 13;
		END_IF
		
	13:
		_MoveParameters[1].targetPosition.x := 120;
		_MoveParameters[1].targetPosition.y := 120;
		_MoveParameters[2].targetPosition.x := 360;
		_MoveParameters[2].targetPosition.y := 120;
		_LocalState := 14;
	
	14:
		FOR _i := 1 TO _MoverCount DO
			_PlanarMover[_i].MoveToPosition
			(
				commandFeedback 	:= _PlanarMoverFeedback[_i],
				targetPosition 		:= _MoveParameters[_i].targetPosition,
				constraint 			:= _MoveParameters[_i].Constraints,
				options 			:= _MoveParameters[_i].Options
			);
		END_FOR
		_LocalState := 15;
	
	15:
		_CommandDone := TRUE;
		FOR _i := 1 TO _MoverCount DO
			IF NOT(_PlanarMoverFeedback[_i].Done) THEN
				_CommandDone := FALSE;
				_InternalCounter := _InternalCounter + 1;
			END_IF
		END_FOR
		
		IF _InternalCounter >= 10000 THEN
			_LocalState := 0;
			_InternalCounter := 0;
			FollowTileEdge := FALSE;
		END_IF
		
		IF _CommandDone THEN
			_CommandDone := FALSE;
			_InternalCounter := 0;
			_LocalState := 16;
		END_IF
		
	16:
		FollowTileEdge := TRUE;
		_LocalState := 0;
		
END_CASE
END_METHOD

METHOD PUBLIC Home : BOOL
VAR_INPUT
END_VAR

// Move movers to the middle of tiles.
	
CASE _LocalState OF
		
	0:
		_LocalState := 1;
		
	1:
		_MoveParameters[1].targetPosition.x := 120;
		_MoveParameters[1].targetPosition.y := 120;
		_MoveParameters[2].targetPosition.x := 360;
		_MoveParameters[2].targetPosition.y := 120;
		_LocalState := 2;
		
	2:
		FOR _i := 1 TO _MoverCount DO
			_PlanarMover[_i].MoveToPosition
			(
				commandFeedback 	:= _PlanarMoverFeedback[_i],
				targetPosition 		:= _MoveParameters[_i].targetPosition,
				constraint 			:= _MoveParameters[_i].Constraints,
				options 			:= _MoveParameters[_i].Options
			);
		END_FOR
		_LocalState := 3;
		
	3:
		_CommandDone := TRUE;
		FOR _i := 1 TO _MoverCount DO
			IF NOT(_PlanarMoverFeedback[_i].Done) THEN
				_CommandDone := FALSE;
				_InternalCounter := _InternalCounter + 1;
			END_IF
		END_FOR
		
		IF _InternalCounter >= 10000 THEN
			_LocalState := 0;
			_InternalCounter := 0;
			Home := FALSE;
		END_IF
		
		IF _CommandDone THEN
			_CommandDone := FALSE;
			_InternalCounter := 0;
			_LocalState := 4;
		END_IF
		
	4:
		Home := TRUE;
		_LocalState := 0;
		
		
END_CASE
END_METHOD

METHOD MeasureWeightOnTile : BOOL
VAR_INPUT
END_VAR

// Measures the weight of an object on a tile
END_METHOD

PROPERTY MoverAcceleration : LREAL
GET
MoverAcceleration := _Acceleration;
END_GET
SET
IF (MoverAcceleration <= 0) OR (MoverAcceleration > 20000) THEN
	_Acceleration := 20000;
ELSE
	_Acceleration := MoverAcceleration;
END_IF
END_SET
END_PROPERTY

PROPERTY MoverBusy : ARRAY [1.._MoverCount] OF BOOL
GET
MoverBusy := _Busy;
END_GET
SET
END_SET
END_PROPERTY

PROPERTY MoverDeceleration : LREAL
GET
MoverDeceleration := _Deceleration;
END_GET
SET
IF (MoverDeceleration <= 0) OR (MoverDeceleration > 20000) THEN
	_Deceleration := 20000;
ELSE
	_Deceleration := MoverDeceleration;
END_IF
END_SET
END_PROPERTY

PROPERTY MoverDone : Array [1.._MoverCount] OF BOOL
GET
MoverDone := _Done;
END_GET
SET
END_SET
END_PROPERTY

PROPERTY MoverEnabled : ARRAY [1.._MoverCount] OF BOOL
GET
MoverEnabled := _Enabled;
END_GET
SET
END_SET
END_PROPERTY

PROPERTY MoverError : ARRAY [1.._MoverCount] OF BOOL
GET
MoverError := _Error;
END_GET
SET
END_SET
END_PROPERTY

PROPERTY MoverJerk : LREAL
GET
MoverJerk := _Jerk;
END_GET
SET
IF (MoverJerk <= 0) OR (MoverJerk > 200000) THEN
	_Jerk := 200000;
ELSE
	_Jerk := MoverJerk;
END_IF
END_SET
END_PROPERTY

PROPERTY MoverLastErrorCode : ARRAY [1.._MoverCount] OF UDINT
GET
MoverLastErrorCode := _ErrorCodePrevious;
END_GET
SET
END_SET
END_PROPERTY

PROPERTY MoverNumberOfRotations : UDINT
GET
MoverNumberOfRotations := _NumberOfRotations;
END_GET
SET
IF (MoverNumberOfRotations < 0) THEN
	_NumberOfRotations := 0;
ELSE
	_NumberOfRotations := MoverNumberOfRotations;
END_IF
END_SET
END_PROPERTY

PROPERTY MoverVelocity : LREAL
GET
MoverVelocity := _Velocity;
END_GET
SET
IF (MoverVelocity <= 0) OR (MoverVelocity > 2000) THEN
	_Velocity := 2000;
ELSE
	_Velocity := MoverVelocity;
END_IF
END_SET
END_PROPERTY

METHOD ResetErrors : BOOL
VAR_INPUT
END_VAR

// Reset errors

CASE _LocalState OF
	
	0: 
		FOR _i := 1 TO _MoverCount DO
			_PlanarMover[_i].Reset(_PlanarMoverFeedback[_i]);
		END_FOR
		_LocalState := 1;
	
	1:	
		_CommandDone := TRUE;
		FOR _i := 1 TO _MoverCount DO
			IF NOT(_PlanarMoverFeedback[_i].Done) THEN
				_CommandDone := FALSE;
				_InternalCounter := _InternalCounter + 1;
			END_IF
		END_FOR
		
		IF _InternalCounter >= 10000 THEN
			_LocalState := 0;
			_InternalCounter := 0;
			ResetErrors := FALSE;
		END_IF
		
		IF _CommandDone THEN
			_CommandDone := FALSE;
			_InternalCounter := 0;
			_LocalState := 2;
		END_IF

			
	2:
		_LocalState := 0;
		_ErrorCount := _ErrorCount + 1;
		ResetErrors := TRUE;
	
END_CASE
END_METHOD

METHOD PUBLIC Spin : BOOL
VAR_INPUT
END_VAR

// Movers spin

CASE _LocalState OF
	
	0:
		_LocalState := 1;

	
	1:
		FOR _i := 1 TO _MoverCount DO
			_PlanarMover[_i].MoveC
			(	
				commandFeedback		:= _PlanarMoverFeedback[_i],
				targetPosition		:= 0,
				constraint			:= _MoveParameters[_i].Constraints,
				options 			:= _MoveParameters[_i].rotateOptions
			);
		END_FOR
		_LocalState := 2;
	
	2:
		_CommandDone := TRUE;
		FOR _i := 1 TO _MoverCount DO
			IF NOT(_PlanarMoverFeedback[_i].Done) THEN
				_CommandDone := FALSE;
				_InternalCounter := _InternalCounter + 1;
			END_IF
		END_FOR
		
		IF _InternalCounter >= 10000 THEN
			_LocalState := 0;
			_InternalCounter := 0;
			Spin := FALSE;
		END_IF
		
		IF _CommandDone THEN
			_CommandDone := FALSE;
			_InternalCounter := 0;
			_LocalState := 3;
		END_IF
		
	3:
		Spin := TRUE;
		_LocalState := 0;
	
END_CASE
END_METHOD

METHOD PUBLIC SwapPlaces : BOOL
VAR_INPUT
END_VAR

// Movers swap tiles, then swap back, then move to home
	
CASE _LocalState OF
	
	0:
		_LocalState := 1;

	1:
		_MoveParameters[1].targetPosition.x := 175;
		_MoveParameters[1].targetPosition.y := 183;
		_MoveParameters[2].targetPosition.x := 301;
		_MoveParameters[2].targetPosition.y := 57;
		_LocalState := 2;
	
	2:
		FOR _i := 1 TO _MoverCount DO
			_PlanarMover[_i].MoveToPosition
			(
				commandFeedback 	:= _PlanarMoverFeedback[_i],
				targetPosition 		:= _MoveParameters[_i].targetPosition,
				constraint 			:= _MoveParameters[_i].Constraints,
				options 			:= _MoveParameters[_i].Options
			);
		END_FOR
		_LocalState := 3;
	
	3:
		_CommandDone := TRUE;
		FOR _i := 1 TO _MoverCount DO
			IF NOT(_PlanarMoverFeedback[_i].Done) THEN
				_CommandDone := FALSE;
				_InternalCounter := _InternalCounter + 1;
			END_IF
		END_FOR
		
		IF _InternalCounter >= 10000 THEN
			_LocalState := 0;
			_InternalCounter := 0;
			SwapPlaces := FALSE;
		END_IF
		
		IF _CommandDone THEN
			_CommandDone := FALSE;
			_InternalCounter := 0;
			_LocalState := 4;
		END_IF

	4:
		_MoveParameters[1].targetPosition.x := 301;
		_MoveParameters[1].targetPosition.y := 183;
		_MoveParameters[2].targetPosition.x := 175;
		_MoveParameters[2].targetPosition.y := 57;
		_LocalState := 5;
	
	5:
		FOR _i := 1 TO _MoverCount DO
			_PlanarMover[_i].MoveToPosition
			(
				commandFeedback 	:= _PlanarMoverFeedback[_i],
				targetPosition 		:= _MoveParameters[_i].targetPosition,
				constraint 			:= _MoveParameters[_i].Constraints,
				options 			:= _MoveParameters[_i].Options
			);
		END_FOR
		_LocalState := 6;
	
	6:
		_CommandDone := TRUE;
		FOR _i := 1 TO _MoverCount DO
			IF NOT(_PlanarMoverFeedback[_i].Done) THEN
				_CommandDone := FALSE;
				_InternalCounter := _InternalCounter + 1;
			END_IF
		END_FOR
		
		IF _InternalCounter >= 10000 THEN
			_LocalState := 0;
			_InternalCounter := 0;
			SwapPlaces := FALSE;
		END_IF
		
		IF _CommandDone THEN
			_CommandDone := FALSE;
			_InternalCounter := 0;
			_LocalState := 7;
		END_IF
		
	7:
		_MoveParameters[1].targetPosition.x := 301;
		_MoveParameters[1].targetPosition.y := 57;
		_MoveParameters[2].targetPosition.x := 175;
		_MoveParameters[2].targetPosition.y := 183;
		_LocalState := 8;
	
	8:
		FOR _i := 1 TO _MoverCount DO
			_PlanarMover[_i].MoveToPosition
			(
				commandFeedback 	:= _PlanarMoverFeedback[_i],
				targetPosition 		:= _MoveParameters[_i].targetPosition,
				constraint 			:= _MoveParameters[_i].Constraints,
				options 			:= _MoveParameters[_i].Options
			);
		END_FOR
		_LocalState := 9;
	
	9:
		_CommandDone := TRUE;
		FOR _i := 1 TO _MoverCount DO
			IF NOT(_PlanarMoverFeedback[_i].Done) THEN
				_CommandDone := FALSE;
				_InternalCounter := _InternalCounter + 1;
			END_IF
		END_FOR
		
		IF _InternalCounter >= 10000 THEN
			_LocalState := 0;
			_InternalCounter := 0;
			SwapPlaces := FALSE;
		END_IF
		
		IF _CommandDone THEN
			_CommandDone := FALSE;
			_InternalCounter := 0;
			_LocalState := 10;
		END_IF
		
	10:
		_MoveParameters[1].targetPosition.x := 175;
		_MoveParameters[1].targetPosition.y := 57;
		_MoveParameters[2].targetPosition.x := 301;
		_MoveParameters[2].targetPosition.y := 183;
		_LocalState := 11;
	
	11:
		FOR _i := 1 TO _MoverCount DO
			_PlanarMover[_i].MoveToPosition
			(
				commandFeedback 	:= _PlanarMoverFeedback[_i],
				targetPosition 		:= _MoveParameters[_i].targetPosition,
				constraint 			:= _MoveParameters[_i].Constraints,
				options 			:= _MoveParameters[_i].Options
			);
		END_FOR
		_LocalState := 12;
	
	12:
		_CommandDone := TRUE;
		FOR _i := 1 TO _MoverCount DO
			IF NOT(_PlanarMoverFeedback[_i].Done) THEN
				_CommandDone := FALSE;
				_InternalCounter := _InternalCounter + 1;
			END_IF
		END_FOR
		
		IF _InternalCounter >= 10000 THEN
			_LocalState := 0;
			_InternalCounter := 0;
			SwapPlaces := FALSE;
		END_IF
		
		IF _CommandDone THEN
			_CommandDone := FALSE;
			_InternalCounter := 0;
			_LocalState := 13;
		END_IF
		
	13:
		_MoveParameters[1].targetPosition.x := 120;
		_MoveParameters[1].targetPosition.y := 120;
		_MoveParameters[2].targetPosition.x := 360;
		_MoveParameters[2].targetPosition.y := 120;
		_LocalState := 14;
	
	14:
		FOR _i := 1 TO _MoverCount DO
			_PlanarMover[_i].MoveToPosition
			(
				commandFeedback 	:= _PlanarMoverFeedback[_i],
				targetPosition 		:= _MoveParameters[_i].targetPosition,
				constraint 			:= _MoveParameters[_i].Constraints,
				options 			:= _MoveParameters[_i].Options
			);
		END_FOR
		_LocalState := 15;
	
	15:
		_CommandDone := TRUE;
		FOR _i := 1 TO _MoverCount DO
			IF NOT(_PlanarMoverFeedback[_i].Done) THEN
				_CommandDone := FALSE;
				_InternalCounter := _InternalCounter + 1;
			END_IF
		END_FOR
		
		IF _InternalCounter >= 10000 THEN
			_LocalState := 0;
			_InternalCounter := 0;
			SwapPlaces := FALSE;
		END_IF
		
		IF _CommandDone THEN
			_CommandDone := FALSE;
			_InternalCounter := 0;
			_LocalState := 16;
		END_IF
		
	16:
		SwapPlaces := TRUE;
		_LocalState := 0;
		
END_CASE
END_METHOD

METHOD PUBLIC Tilt : BOOL
VAR_INPUT
END_VAR

// Movers tilt

CASE _LocalState OF
	
	0:
		_LocalState := 1;
		
	1:
		FOR _i := 1 TO _MoverCount DO
			_PlanarMover[_i].MoveZ
			(	
				commandFeedback		:= _PlanarMoverFeedback[_i],
				targetPosition		:= 5.0,
				constraint			:= _MoveParameters[_i].Constraints
			);
		END_FOR
		_LocalState := 2;
	
	2:
		_CommandDone := TRUE;
		FOR _i := 1 TO _MoverCount DO
			IF NOT(_PlanarMoverFeedback[_i].Done) THEN
				_CommandDone := FALSE;
				_InternalCounter := _InternalCounter + 1;
			END_IF
		END_FOR
		
		IF _InternalCounter >= 10000 THEN
			_LocalState := 0;
			_InternalCounter := 0;
			Tilt := FALSE;
		END_IF
		
		IF _CommandDone THEN
			_CommandDone := FALSE;
			_InternalCounter := 0;
			_LocalState := 3;
		END_IF

	
	3:
		FOR _i := 1 TO _MoverCount DO
			_PlanarMover[_i].MoveA
			(	
				commandFeedback		:= _PlanarMoverFeedback[_i],
				targetPosition		:= 4.0,
				constraint			:= _MoveParameters[_i].Constraints
			);
		END_FOR
		_LocalState := 4;
	
	4:
		_CommandDone := TRUE;
		FOR _i := 1 TO _MoverCount DO
			IF NOT(_PlanarMoverFeedback[_i].Done) THEN
				_CommandDone := FALSE;
				_InternalCounter := _InternalCounter + 1;
			END_IF
		END_FOR
		
		IF _InternalCounter >= 10000 THEN
			_LocalState := 0;
			_InternalCounter := 0;
			Tilt := FALSE;
		END_IF
		
		IF _CommandDone THEN
			_CommandDone := FALSE;
			_InternalCounter := 0;
			_LocalState := 5;
		END_IF
		
	5:
		FOR _i := 1 TO _MoverCount DO
			_PlanarMover[_i].MoveA
			(	
				commandFeedback		:= _PlanarMoverFeedback[_i],
				targetPosition		:= -4.0,
				constraint			:= _MoveParameters[_i].Constraints
			);
		END_FOR
		_LocalState := 6;
	
	6:
		_CommandDone := TRUE;
		FOR _i := 1 TO _MoverCount DO
			IF NOT(_PlanarMoverFeedback[_i].Done) THEN
				_CommandDone := FALSE;
				_InternalCounter := _InternalCounter + 1;
			END_IF
		END_FOR
		
		IF _InternalCounter >= 10000 THEN
			_LocalState := 0;
			_InternalCounter := 0;
			Tilt := FALSE;
		END_IF
		
		IF _CommandDone THEN
			_CommandDone := FALSE;
			_InternalCounter := 0;
			_LocalState := 7;
		END_IF
	
	7:
		FOR _i := 1 TO _MoverCount DO
			_PlanarMover[_i].MoveA
			(	
				commandFeedback		:= _PlanarMoverFeedback[_i],
				targetPosition		:= 0.0,
				constraint			:= _MoveParameters[_i].Constraints
			);
		END_FOR
		_LocalState := 8;
	
	8:
		_CommandDone := TRUE;
		FOR _i := 1 TO _MoverCount DO
			IF NOT(_PlanarMoverFeedback[_i].Done) THEN
				_CommandDone := FALSE;
				_InternalCounter := _InternalCounter + 1;
			END_IF
		END_FOR
		
		IF _InternalCounter >= 10000 THEN
			_LocalState := 0;
			_InternalCounter := 0;
			Tilt := FALSE;
		END_IF
		
		IF _CommandDone THEN
			_CommandDone := FALSE;
			_InternalCounter := 0;
			_LocalState := 9;
		END_IF
		
	9:
		FOR _i := 1 TO _MoverCount DO
			_PlanarMover[_i].MoveB
			(	
				commandFeedback		:= _PlanarMoverFeedback[_i],
				targetPosition		:= 4.0,
				constraint			:= _MoveParameters[_i].Constraints
			);
		END_FOR
		_LocalState := 10;
	
	10:
		_CommandDone := TRUE;
		FOR _i := 1 TO _MoverCount DO
			IF NOT(_PlanarMoverFeedback[_i].Done) THEN
				_CommandDone := FALSE;
				_InternalCounter := _InternalCounter + 1;
			END_IF
		END_FOR
		
		IF _InternalCounter >= 10000 THEN
			_LocalState := 0;
			_InternalCounter := 0;
			Tilt := FALSE;
		END_IF
		
		IF _CommandDone THEN
			_CommandDone := FALSE;
			_InternalCounter := 0;
			_LocalState := 11;
		END_IF
		
	11:
		FOR _i := 1 TO _MoverCount DO
			_PlanarMover[_i].MoveB
			(	
				commandFeedback		:= _PlanarMoverFeedback[_i],
				targetPosition		:= -4.0,
				constraint			:= _MoveParameters[_i].Constraints
			);
		END_FOR
		_LocalState := 12;
	
	12:
		_CommandDone := TRUE;
		FOR _i := 1 TO _MoverCount DO
			IF NOT(_PlanarMoverFeedback[_i].Done) THEN
				_CommandDone := FALSE;
				_InternalCounter := _InternalCounter + 1;
			END_IF
		END_FOR
		
		IF _InternalCounter >= 10000 THEN
			_LocalState := 0;
			_InternalCounter := 0;
			Tilt := FALSE;
		END_IF
		
		IF _CommandDone THEN
			_CommandDone := FALSE;
			_InternalCounter := 0;
			_LocalState := 13;
		END_IF
	
	13:
		FOR _i := 1 TO _MoverCount DO
			_PlanarMover[_i].MoveB
			(	
				commandFeedback		:= _PlanarMoverFeedback[_i],
				targetPosition		:= 0.0,
				constraint			:= _MoveParameters[_i].Constraints
			);
		END_FOR
		_LocalState := 14;
	
	14:
		_CommandDone := TRUE;
		FOR _i := 1 TO _MoverCount DO
			IF NOT(_PlanarMoverFeedback[_i].Done) THEN
				_CommandDone := FALSE;
				_InternalCounter := _InternalCounter + 1;
			END_IF
		END_FOR
		
		IF _InternalCounter >= 10000 THEN
			_LocalState := 0;
			_InternalCounter := 0;
			Tilt := FALSE;
		END_IF
		
		IF _CommandDone THEN
			_CommandDone := FALSE;
			_InternalCounter := 0;
			_LocalState := 15;
		END_IF
		
	15:
		FOR _i := 1 TO _MoverCount DO
			_PlanarMover[_i].MoveZ
			(	
				commandFeedback		:= _PlanarMoverFeedback[_i],
				targetPosition		:= 2.0,
				constraint			:= _MoveParameters[_i].Constraints
			);
		END_FOR
		_LocalState := 16;
	
	16:
		_CommandDone := TRUE;
		FOR _i := 1 TO _MoverCount DO
			IF NOT(_PlanarMoverFeedback[_i].Done) THEN
				_CommandDone := FALSE;
				_InternalCounter := _InternalCounter + 1;
			END_IF
		END_FOR
		
		IF _InternalCounter >= 10000 THEN
			_LocalState := 0;
			_InternalCounter := 0;
			Tilt := FALSE;
		END_IF
		
		IF _CommandDone THEN
			_CommandDone := FALSE;
			_InternalCounter := 0;
			_LocalState := 17;
		END_IF
		
	17:
		Tilt := TRUE;
		_LocalState := 0;
	
END_CASE
END_METHOD

METHOD PUBLIC VaryMoverHeight : BOOL
VAR_INPUT
END_VAR

// Movers vary their height multiple times

CASE _LocalState OF
	
	0:
		_LocalState := 1;
	
	1:
		FOR _i := 1 TO _MoverCount DO
			_PlanarMover[_i].MoveZ
			(	
				commandFeedback		:= _PlanarMoverFeedback[_i],
				targetPosition		:= 5.0,
				constraint			:= _MoveParameters[_i].Constraints
			);
		END_FOR
		_LocalState := 2;
	
	2:
		_CommandDone := TRUE;
		FOR _i := 1 TO _MoverCount DO
			IF NOT(_PlanarMoverFeedback[_i].Done) THEN
				_CommandDone := FALSE;
				_InternalCounter := _InternalCounter + 1;
			END_IF
		END_FOR
		
		IF _InternalCounter >= 10000 THEN
			_LocalState := 0;
			_InternalCounter := 0;
			VaryMoverHeight := FALSE;
		END_IF
		
		IF _CommandDone THEN
			_CommandDone := FALSE;
			_InternalCounter := 0;
			_LocalState := 3;
		END_IF
		
	3:
		FOR _i := 1 TO _MoverCount DO
			_PlanarMover[_i].MoveZ
			(	
				commandFeedback		:= _PlanarMoverFeedback[_i],
				targetPosition		:= 2.0,
				constraint			:= _MoveParameters[_i].Constraints
			);
		END_FOR
		_LocalState := 4;
	
	4:
		_CommandDone := TRUE;
		FOR _i := 1 TO _MoverCount DO
			IF NOT(_PlanarMoverFeedback[_i].Done) THEN
				_CommandDone := FALSE;
				_InternalCounter := _InternalCounter + 1;
			END_IF
		END_FOR
		
		IF _InternalCounter >= 10000 THEN
			_LocalState := 0;
			_InternalCounter := 0;
			VaryMoverHeight := FALSE;
		END_IF
		
		IF _CommandDone THEN
			_CommandDone := FALSE;
			_InternalCounter := 0;
			_LocalState := 5;
		END_IF
		
	5:
		FOR _i := 1 TO _MoverCount DO
			_PlanarMover[_i].MoveZ
			(	
				commandFeedback		:= _PlanarMoverFeedback[_i],
				targetPosition		:= 5.0,
				constraint			:= _MoveParameters[_i].Constraints
			);
		END_FOR
		_LocalState := 6;
	
	6:
		_CommandDone := TRUE;
		FOR _i := 1 TO _MoverCount DO
			IF NOT(_PlanarMoverFeedback[_i].Done) THEN
				_CommandDone := FALSE;
				_InternalCounter := _InternalCounter + 1;
			END_IF
		END_FOR
		
		IF _InternalCounter >= 10000 THEN
			_LocalState := 0;
			_InternalCounter := 0;
			VaryMoverHeight := FALSE;
		END_IF
		
		IF _CommandDone THEN
			_CommandDone := FALSE;
			_InternalCounter := 0;
			_LocalState := 7;
		END_IF
		
	7:
		FOR _i := 1 TO _MoverCount DO
			_PlanarMover[_i].MoveZ
			(	
				commandFeedback		:= _PlanarMoverFeedback[_i],
				targetPosition		:= 2.0,
				constraint			:= _MoveParameters[_i].Constraints
			);
		END_FOR
		_LocalState := 8;
	
	8:
		_CommandDone := TRUE;
		FOR _i := 1 TO _MoverCount DO
			IF NOT(_PlanarMoverFeedback[_i].Done) THEN
				_CommandDone := FALSE;
				_InternalCounter := _InternalCounter + 1;
			END_IF
		END_FOR
		
		IF _InternalCounter >= 10000 THEN
			_LocalState := 0;
			_InternalCounter := 0;
			VaryMoverHeight := FALSE;
		END_IF
		
		IF _CommandDone THEN
			_CommandDone := FALSE;
			_InternalCounter := 0;
			_LocalState := 9;
		END_IF
		
	9:
		FOR _i := 1 TO _MoverCount DO
			_PlanarMover[_i].MoveZ
			(	
				commandFeedback		:= _PlanarMoverFeedback[_i],
				targetPosition		:= 5.0,
				constraint			:= _MoveParameters[_i].Constraints
			);
		END_FOR
		_LocalState := 10;
	
	10:
		_CommandDone := TRUE;
		FOR _i := 1 TO _MoverCount DO
			IF NOT(_PlanarMoverFeedback[_i].Done) THEN
				_CommandDone := FALSE;
				_InternalCounter := _InternalCounter + 1;
			END_IF
		END_FOR
		
		IF _InternalCounter >= 10000 THEN
			_LocalState := 0;
			_InternalCounter := 0;
			VaryMoverHeight := FALSE;
		END_IF
		
		IF _CommandDone THEN
			_CommandDone := FALSE;
			_InternalCounter := 0;
			_LocalState := 11;
		END_IF

	11:
		FOR _i := 1 TO _MoverCount DO
			_PlanarMover[_i].MoveZ
			(	
				commandFeedback		:= _PlanarMoverFeedback[_i],
				targetPosition		:= 2.0,
				constraint			:= _MoveParameters[_i].Constraints
			);
		END_FOR
		_LocalState := 12;
	
	12:
		_CommandDone := TRUE;
		FOR _i := 1 TO _MoverCount DO
			IF NOT(_PlanarMoverFeedback[_i].Done) THEN
				_CommandDone := FALSE;
				_InternalCounter := _InternalCounter + 1;
			END_IF
		END_FOR
		
		IF _InternalCounter >= 10000 THEN
			_LocalState := 0;
			_InternalCounter := 0;
			VaryMoverHeight := FALSE;
		END_IF
		
		IF _CommandDone THEN
			_CommandDone := FALSE;
			_InternalCounter := 0;
			_LocalState := 13;
		END_IF
		
	13:
		VaryMoverHeight := TRUE;
		_LocalState := 0;

END_CASE
END_METHOD

END_FUNCTION_BLOCK

// ---- POUs/Analytics/CoeToPlc.TcPOU
PROGRAM CoeToPlc
VAR
	
	CoeTrigger		: TON;
	CoeTriggerTime	: TIME := T#50MS;
	
	TileTemp1		: FB_EcCoESdoRead;
	Temperature1	: WORD;
	
	TileTemp2		: FB_EcCoESdoRead;
	Temperature2	: WORD;
			
	FanSpeed1		: FB_EcCoESdoRead;
	Speed1			: BYTE;
	
	FanSpeed2		: FB_EcCoESdoRead;
	Speed2			: BYTE;
	
END_VAR



CoeTrigger(IN := NOT(CoeTrigger.Q), PT := CoeTriggerTime);


TileTemp1
(
    sNetId     := '192.168.5.90.7.1',
    nSlaveAddr := 1001,
    nIndex     := 16#FA00,
    nSubIndex  := 25,
    pDstBuf    := ADR(Temperature1),
    cbBufLen   := SIZEOF(Temperature1),
    bExecute   := CoeTrigger.Q
);

TileTemp2
(
    sNetId     := '192.168.5.90.7.1',
    nSlaveAddr := 1003,
    nIndex     := 16#FA00,
    nSubIndex  := 25,
    pDstBuf    := ADR(Temperature2),
    cbBufLen   := SIZEOF(Temperature2),
    bExecute   := CoeTrigger.Q
);

FanSpeed1
(
    sNetId     := '192.168.5.90.7.1',
    nSlaveAddr := 1001,
    nIndex     := 16#FA00,
    nSubIndex  := 28,
    pDstBuf    := ADR(Speed1),
    cbBufLen   := SIZEOF(Speed1),
    bExecute   := CoeTrigger.Q
);

FanSpeed2
(
    sNetId     := '192.168.5.90.7.1',
    nSlaveAddr := 1003,
    nIndex     := 16#FA00,
    nSubIndex  := 28,
    pDstBuf    := ADR(Speed2),
    cbBufLen   := SIZEOF(Speed2),
    bExecute   := CoeTrigger.Q
);

END_PROGRAM

// ---- VISUs/Visualization.TcVIS
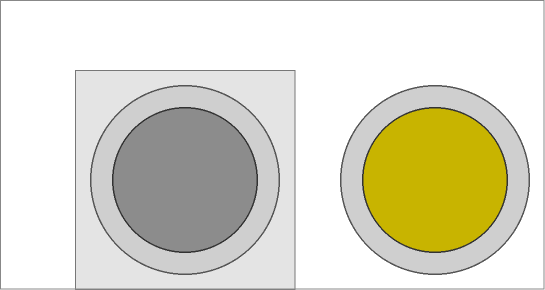
VISUALIZATION Visualization  // 545x290
    PushSwitch (75,70 220x220), variable: IO.HardwareInput[1], behaviour: TAP, style: Switch-PushSwitch-Gray
    Lamp1 (325,70 220x220), variable: IO.HardwareOutput[1], style: Lamp-Lamp1-Yellow
END_VISUALIZATION
